(* IEC 61131-3 sources: BODAS-HelloWorld/extracted_st/bodas_rc18_12_40/plc_logic/application/02_easyconfig/easyconfig_import/bds_sent_ec/bds_sent_ec_gvl, 1 file *)

(* ---- bds_sent_ec_gvl.st ---- *)
(* --- Interface --- *)
{attribute 'qualified_only' := ''}
VAR_GLOBAL CONSTANT
    bds_sent_postVariants_du8      : USINT := 1;
    bds_sent_maxDataNibbles_du8    : USINT := 6;
    bds_sent_rxFastDataBufSize_du8 : USINT := 0;
    bds_sent_rxSlowDataBufSize_du8 : USINT := 0;
END_VAR
